FUNCTION_BLOCK NeredaCapacitySpToDBlowersSp (* Basic Function Block Type *)
  (* Standard: 61499-2 *)
  (* Version 0.0, 10/7/2023, SESA685388, Schneider Electric, Template *)
  PACKAGE SE.Nereda;
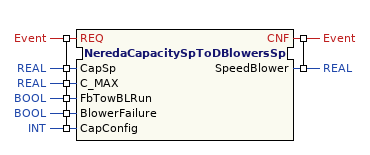
  EVENT_INPUT
    REQ WITH CapSp, C_MAX, FbTowBLRun, BlowerFailure, CapConfig;
  END_EVENT
  EVENT_OUTPUT
    CNF WITH SpeedBlower; (* Execution Confirmation *)
  END_EVENT
  VAR_INPUT
    CapSp : REAL; (* Input event qualifier *)
    C_MAX : REAL;
    FbTowBLRun : BOOL;
    BlowerFailure : BOOL;
    CapConfig : INT;
  END_VAR
  VAR_OUTPUT
    SpeedBlower : REAL;
  END_VAR
  VAR
    Equal : BOOL;
  END_VAR
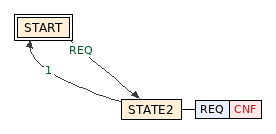
  EC_STATES
    START; (* Initial State *)
    STATE2 : REQ -> CNF;
  END_STATES
  EC_TRANSITIONS
    START TO STATE2 := REQ;
    STATE2 TO START := 1;
  END_TRANSITIONS
  ALGORITHM REQ IN ST: (* Initialization algorithm *)
;
IF CapSp > 0 AND CapSp <= C_MAX AND NOT FbTowBLRun THEN
	SpeedBlower := (CapSp / C_MAX) * 100;
END_IF;

IF C_MAX < CapSp AND CapSp <= 100.00 AND FbTowBLRun THEN
	IF NOT BlowerFailure THEN
		IF CapConfig = 1 THEN
			SpeedBlower := ((CapSp - C_MAX) / (100.00 - C_MAX)) * 86.00; //0% - 86%
		ELSIF CapConfig = 2 THEN
			SpeedBlower := 50.00 + ((CapSp - C_MAX) / (100.00 - C_MAX)) * (86.00 - 50.00); // 50% - 86%
		END_IF;
	ELSE
		SpeedBlower := CapSp; //To check this senario with Nereda Teams
	END_IF;
END_IF;

IF CapSp = 0 THEN
	SpeedBlower := 0.00;
END_IF;
  END_ALGORITHM
END_FUNCTION_BLOCK
